Staubli VAL3: DebV2.dtx

mdesc mNomSpeed
jointRx jJointRx[2]
  [1] = {j1=180}
dio SortiePower = {link=POWERLINK-1\%Q1}
dio EntreePower = {link=POWERLINK-1\%I0}
tool tTool = {z=50, fatherId=flange[0], ioLink=valve1}
